(* PLC project Generated.project, CODESYS CODESYS V3.5 SP19 Patch 1 *)
(* stored: creationDateTime 2026-08-18T12:52:51.318285, modificationDateTime 2026-08-18T12:52:51.318285 *)

(* ═══════════════════════════════════════════════════════════════ ⚙️ ST_SyncHMI — Données d'échange IHM pour la synchronisation M1/M2 ─────────────────────────────────────────────────────────────── 📄 Structuration en Cmd / State / Cfg / Bypass , homogène avec ST_WinchHMI. ═══════════════════════════════════════════════════════════════ *)
TYPE ST_SyncHMI : STRUCT
  Cmd : ST_SyncCmd;
  State : ST_SyncState;
  Cfg : ST_SyncCfg;
  Bypass : ST_BypassSync;
END_STRUCT;
END_TYPE

(* ═══════════════════════════════════════════════════════════════ ST_BypassSync — Bypass de la surveillance synchronisation M1/M2 🔒 Doctrine : actionnable UNIQUEMENT en MAINT_N2, RETAIN, jamais masque les autres défauts du même bloc (voir REGISTRE_ACTIONS_Bypass_v1.0 (archive)). ═══════════════════════════════════════════════════════════════ *)
TYPE ST_BypassSync : STRUCT
  Global : BOOL := FALSE;  (* 🌐 Bypass GLOBAL synchro : ignore toute erreur de synchronisation *)
  Initialized : BOOL := FALSE;  (* 🚦 flag restauration boot *)
END_STRUCT;
END_TYPE

(* ═══════════════════════════════════════════════════════════════ ST_SyncCfg — Configuration de la synchronisation M1/M2 ═══════════════════════════════════════════════════════════════ *)
TYPE ST_SyncCfg : STRUCT
  CfgSyncTolerance_M : REAL := 0.8;  (* 📐 Tolérance max d'écart (m) — Dégradation Palier 1 dès 0.8m *)
  Initialized : BOOL := FALSE;  (* 🚦 flag restauration boot, ex-CfgInitialized renommé pour cohérence avec ST_WinchCfg *)
END_STRUCT;
END_TYPE

(* ═══════════════════════════════════════════════════════════════ 🎮 ST_SyncCmd — Commandes IHM pour la synchronisation M1/M2 ═══════════════════════════════════════════════════════════════ *)
TYPE ST_SyncCmd : STRUCT
  SelSyncEnable : BOOL := TRUE;  (* ☑️ coché = synchro voulue (MAINT_N1/N2), ex-OverrideSync inversé *)
END_STRUCT;
END_TYPE

(* ═══════════════════════════════════════════════════════════════ 🚦 ST_SyncState — États et diagnostics de la synchronisation M1/M2 ═══════════════════════════════════════════════════════════════ *)
TYPE ST_SyncState : STRUCT
  DeltaPos_M : REAL;  (* 📊 Écart de position réel mesuré (m) *)
  SyncActive : BOOL;  (* ⚖️ Indicateur si surveillance active *)
  SyncWarn : BOOL;  (* ⚠️ LED d'alarme écart hors tolérance *)
  SyncDegradedStep1 : BOOL;  (* 🐢 Écart modéré actif : limitation forcée au Palier 1 *)
  Ready : BOOL;  (* 🟢 Bloc de synchro prêt *)
  Error : BOOL;  (* Alarme synchro active *)
  ErrorId : WORD;  (* ❌ Code défaut synchro *)
  FBState : E_State;  (* 🤖 État de l'automate interne (FB_WinchSync) — ex-"State", renommé pour éviter collision avec le sous-struct State *)
END_STRUCT;
END_TYPE

(* values of E_State: DISABLED: Enable faux, neutralisé; INIT: Démarrage / vérifs; READY: Prêt, attend ordre; BUSY: Action en cours; DONE: Action terminée; STOPPING: Décél rampe avant arrêt (StartStop=FALSE ou SafeStop=TRUE) *)

{attribute 'qualified_only'}
{attribute 'strict'}
TYPE E_State : (DISABLED := 0, INIT := 1, READY := 2, BUSY := 3, DONE := 4, STOPPING := 5);
END_TYPE
